TYPE TcoDaqData :
STRUCT
	_s : STRING;
	_i : INT;
END_STRUCT
END_TYPE

(* stored: Version 1.1.0.1
   DUT TcoDaqData: Id {92e7033b-5043-0e97-09b7-ad1688754aec} *)
